(* CODESYS project e!C_VisuTrend_Test_1.ecp

Project tree, tasks and I/O mapping:
  Controller : 750-8202 PFC200 2ETH RS, WAGO, order no. 0750-8202, version 5.11.1.16
    application Application
      libraries: 
      task PLC_Task (cyclic, interval t#10ms, priority 14) calls PLC_PRG
      task VISU_TASK (cyclic, interval 100 ms, priority 15) calls VisuElems.Visu_Prg
      task TrendRecordingTask (cyclic, interval 100 ms, priority 15) calls VisuTrendStorageAccess.GlobalInstances.g_TrendRecordingManager.CyclicCall
      program PLC_PRG [ST]
      visualisation Visualization
      Trend Recording Manager
        Visualization_Trend1
    DeviceAdapter
    Kbus : Kbus, WAGO, version 1.4.0.2
        unmapped channels: K-BUS diagnostics
    MODBUS
      MODBUS : MODBUS, WAGO, order no. n/a, version 1.1.1.15
    Serial
      COM1 : COM1, WAGO, version 0.0.0.19
  libraries: VisuSymbols, 3.5.10.0 (System); WagoVisuIcons, 1.0.0.8 (WAGO)
  text list GlobalTextList
*)

// Controller/Application/PLC_PRG
PROGRAM PLC_PRG
VAR
	rTrendVar1: REAL;
	rSineTest: REAL;
	rSineTestDelta: REAL := 0.01;
END_VAR




rSineTest := rSineTest + rSineTestDelta;
IF (rSineTest >= (2*3.14)) THEN
	rSineTest := 0;
END_IF

rTrendVar1 := 100 + (100*SIN(rSineTest));

END_PROGRAM

// Controller/Application/Visualization
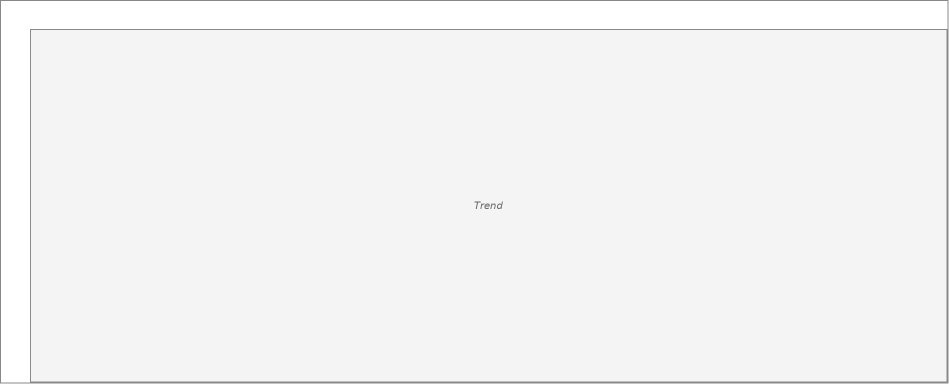
VISUALIZATION Visualization  // 949x384
    Trend (30,29 917x353)
        p758368661: M/d/yyyy
        p2423372160: h:mm:ss tt:ms
        p2833066001: Visualization_Trend1
END_VISUALIZATION
